// TIA Portal V20 export
TYPE "IO_Device_Functinal_Test"
   STRUCT
      Life_Trigger_PLC_Functional_Test_1 : Bool;
      Star_Test_PLC_Functional_Test_1 : Bool;
      Button_PLC_Functional_Test_1 : Bool;
      Electrical_Current_Test_Approved_PLC_Functional_Test_1 : Bool;
      Visual_Test_Approved_PLC_Functional_Test_1 : Bool;
      Electrical_Current_Read_PLC_Functional_Test_1 : UInt;
      Life_Trigger_PLC_Functional_Test_3 : Bool;
      Star_Test_PLC_Functional_Test_3 : Bool;
      Button_PLC_Functional_Test_3 : Bool;
      Electrical_Current_Test_Approved_PLC_Functional_Test_3 : Bool;
      Visual_Test_Approved_PLC_Functional_Test_3 : Bool;
      Electrical_Current_Read_PLC_Functional_Test_3 : UInt;
      Life_Trigger_PLC_Functional_Test_5 : Bool;
      Star_Test_PLC_Functional_Test_5 : Bool;
      Button_PLC_Functional_Test_5 : Bool;
      Electrical_Current_Test_Approved_PLC_Functional_Test_5 : Bool;
      Visual_Test_Approved_PLC_Functional_Test_5 : Bool;
      Electrical_Current_Read_PLC_Functional_Test_5 : UInt;
      Life_Trigger_PLC_Functional_Test_7 : Bool;
      Star_Test_PLC_Functional_Test_7 : Bool;
      Button_PLC_Functional_Test_7 : Bool;
      Electrical_Current_Test_Approved_PLC_Functional_Test_7 : Bool;
      Visual_Test_Approved_PLC_Functional_Test_7 : Bool;
      Electrical_Current_Read_PLC_Functional_Test_7 : UInt;
      Life_Trigger_PLC_Functional_Test_9 : Bool;
      Star_Test_PLC_Functional_Test_9 : Bool;
      Button_PLC_Functional_Test_9 : Bool;
      Electrical_Current_Test_Approved_PLC_Functional_Test_9 : Bool;
      Visual_Test_Approved_PLC_Functional_Test_9 : Bool;
      Electrical_Current_Read_PLC_Functional_Test_9 : UInt;
      Life_Trigger_PLC_Functional_Test_11 : Bool;
      Star_Test_PLC_Functional_Test_11 : Bool;
      Button_PLC_Functional_Test_11 : Bool;
      Electrical_Current_Test_Approved_PLC_Functional_Test_11 : Bool;
      Visual_Test_Approved_PLC_Functional_Test_11 : Bool;
      Electrical_Current_Read_PLC_Functional_Test_11 : UInt;
      Life_Trigger_PLC_Functional_Test_13 : Bool;
      Star_Test_PLC_Functional_Test_13 : Bool;
      Button_PLC_Functional_Test_13 : Bool;
      Electrical_Current_Test_Approved_PLC_Functional_Test_13 : Bool;
      Visual_Test_Approved_PLC_Functional_Test_13 : Bool;
      Electrical_Current_Read_PLC_Functional_Test_13 : UInt;
      Life_Trigger_PLC_Functional_Test_15 : Bool;
      Star_Test_PLC_Functional_Test_15 : Bool;
      Button_PLC_Functional_Test_15 : Bool;
      Electrical_Current_Test_Approved_PLC_Functional_Test_15 : Bool;
      Visual_Test_Approved_PLC_Functional_Test_15 : Bool;
      Electrical_Current_Read_PLC_Functional_Test_15 : UInt;
      Life_Trigger_PLC_Functional_Test_17 : Bool;
      Star_Test_PLC_Functional_Test_17 : Bool;
      Button_PLC_Functional_Test_17 : Bool;
      Electrical_Current_Test_Approved_PLC_Functional_Test_17 : Bool;
      Visual_Test_Approved_PLC_Functional_Test_17 : Bool;
      Electrical_Current_Read_PLC_Functional_Test_17 : UInt;
      Life_Trigger_PLC_Functional_Test_19 : Bool;
      Star_Test_PLC_Functional_Test_19 : Bool;
      Button_PLC_Functional_Test_19 : Bool;
      Electrical_Current_Test_Approved_PLC_Functional_Test_19 : Bool;
      Visual_Test_Approved_PLC_Functional_Test_19 : Bool;
      Electrical_Current_Read_PLC_Functional_Test_19 : UInt;
      Life_Trigger_PLC_Functional_Test_21 : Bool;
      Star_Test_PLC_Functional_Test_21 : Bool;
      Button_PLC_Functional_Test_21 : Bool;
      Electrical_Current_Test_Approved_PLC_Functional_Test_21 : Bool;
      Visual_Test_Approved_PLC_Functional_Test_21 : Bool;
      Electrical_Current_Read_PLC_Functional_Test_21 : UInt;
      Life_Trigger_PLC_Functional_Test_23 : Bool;
      Star_Test_PLC_Functional_Test_23 : Bool;
      Button_PLC_Functional_Test_23 : Bool;
      Electrical_Current_Test_Approved_PLC_Functional_Test_23 : Bool;
      Visual_Test_Approved_PLC_Functional_Test_23 : Bool;
      Electrical_Current_Read_PLC_Functional_Test_23 : UInt;
      Life_Trigger_PLC_Functional_Test_25 : Bool;
      Star_Test_PLC_Functional_Test_25 : Bool;
      Button_PLC_Functional_Test_25 : Bool;
      Electrical_Current_Test_Approved_PLC_Functional_Test_25 : Bool;
      Visual_Test_Approved_PLC_Functional_Test_25 : Bool;
      Electrical_Current_Read_PLC_Functional_Test_25 : UInt;
      Life_Trigger_PLC_Functional_Test_27 : Bool;
      Star_Test_PLC_Functional_Test_27 : Bool;
      Button_PLC_Functional_Test_27 : Bool;
      Electrical_Current_Test_Approved_PLC_Functional_Test_27 : Bool;
      Visual_Test_Approved_PLC_Functional_Test_27 : Bool;
      Electrical_Current_Read_PLC_Functional_Test_27 : UInt;
      Life_Trigger_PLC_Functional_Test_29 : Bool;
      Star_Test_PLC_Functional_Test_29 : Bool;
      Button_PLC_Functional_Test_29 : Bool;
      Electrical_Current_Test_Approved_PLC_Functional_Test_29 : Bool;
      Visual_Test_Approved_PLC_Functional_Test_29 : Bool;
      Electrical_Current_Read_PLC_Functional_Test_29 : UInt;
   END_STRUCT;
END_TYPE
